(* IEC 61131-3 sources: IEC61131-3-CDSV3/Math Expressions Evaluator/src/20 Program Organization Units/_Internal, 7 files *)

(* ---- FuEvaluateFunctionCall.pou ---- *)
(*#-#-#-#-#-#-#-#-#-#---Declaration---#-#-#-#-#-#-#-#-#-#-#-#-#*)

// Evaluates a function call.
// First all necessary arguments are resolved to LREAL and then the function gets executed.
// The return value will indicate a successful evaluation.
{attribute 'qualified_only'}
FUNCTION INTERNAL FuEvaluateFunctionCall : BOOL
VAR_INPUT
    typFunctionToken: typExpressionToken;
    uiMaxCursor: UINT;
END_VAR
VAR_IN_OUT
    atTokens: ARRAY [*] OF typExpressionToken;
    uiCursor: UINT;

    alrVariables: ARRAY [*] OF LREAL;
    alrInternalVariables: ARRAY [*] OF LREAL;
END_VAR
VAR_OUTPUT
    lrResult: LREAL;
    sError: STRING;
END_VAR
{library PRIVATE}
VAR
    i: UINT;
    j: UINT;

    tempArgs: ARRAY [0..8] OF LREAL;
    tempHelperValue: LREAL;
END_VAR
VAR CONSTANT
    CONST_PI: LREAL := 3.14159265359;
END_VAR
(*#-#-#-#-#-#-#-#-#-#---Implementation---#-#-#-#-#-#-#-#-#-#-#-#-#*)

IF typFunctionToken.eType <> eTokenType.FUNCTION_CALL THEN
    sError := Standard.CONCAT('Invalid function call token at ', TO_STRING(uiCursor));
    RETURN;
END_IF

IF uiCursor + typFunctionToken.uiArgsCount > uiMaxCursor THEN
    sError := Standard.CONCAT('Not enough arguments for function call at ', TO_STRING(uiCursor));
    RETURN;
END_IF

FOR i := 0 TO (typFunctionToken.uiArgsCount - 1) BY 1 DO
    j := uiCursor + i + 1;

    IF NOT FuEvaluateTokenSingle(atTokens[j], j, alrVariables, alrInternalVariables, lrResult => tempArgs[i], sError => sError) THEN
        RETURN;
    END_IF
END_FOR

uiCursor := uiCursor + typFunctionToken.uiArgsCount;

IF typFunctionToken.sIdentifier = Constants.FUN_ABS THEN
    FuEvaluateFunctionCall := TRUE;
    lrResult := ABS(tempArgs[0]);
ELSIF typFunctionToken.sIdentifier = Constants.FUN_ACOS THEN
    FuEvaluateFunctionCall := TRUE;
    lrResult := ACOS(tempArgs[0]);
ELSIF typFunctionToken.sIdentifier = Constants.FUN_ASIN THEN
    FuEvaluateFunctionCall := TRUE;
    lrResult := ASIN(tempArgs[0]);
ELSIF typFunctionToken.sIdentifier = Constants.FUN_ATAN THEN
    FuEvaluateFunctionCall := TRUE;
    lrResult := ATAN(tempArgs[0]);
ELSIF typFunctionToken.sIdentifier = Constants.FUN_CEIL THEN
    FuEvaluateFunctionCall := TRUE;
    lrResult := FPU.Ceil(tempArgs[0]);
ELSIF typFunctionToken.sIdentifier = Constants.FUN_COS THEN
    FuEvaluateFunctionCall := TRUE;
    lrResult := COS(tempArgs[0]);
ELSIF typFunctionToken.sIdentifier = Constants.FUN_DEG THEN
    FuEvaluateFunctionCall := TRUE;
    lrResult := tempArgs[0] * 180 / CONST_PI;
ELSIF typFunctionToken.sIdentifier = Constants.FUN_FLOOR THEN
    FuEvaluateFunctionCall := TRUE;
    lrResult := FPU.Floor(tempArgs[0]);
ELSIF typFunctionToken.sIdentifier = Constants.FUN_LOG THEN
    FuEvaluateFunctionCall := TRUE;
    lrResult := LOG(tempArgs[0]);
ELSIF typFunctionToken.sIdentifier = Constants.FUN_LN THEN
    FuEvaluateFunctionCall := TRUE;
    lrResult := LN(tempArgs[0]);
ELSIF typFunctionToken.sIdentifier = Constants.FUN_RAD THEN
    FuEvaluateFunctionCall := TRUE;
    lrResult := tempArgs[0] * CONST_PI / 180;
ELSIF typFunctionToken.sIdentifier = Constants.FUN_ROUND THEN
    FuEvaluateFunctionCall := TRUE;

    IF (tempArgs[0] - FPU.Truncate(tempArgs[0])) >= 0.5 THEN
        lrResult := FPU.Ceil(tempArgs[0]);
    ELSE
        lrResult := FPU.Floor(tempArgs[0]);
    END_IF
ELSIF typFunctionToken.sIdentifier = Constants.FUN_SIN THEN
    FuEvaluateFunctionCall := TRUE;
    lrResult := SIN(tempArgs[0]);
ELSIF typFunctionToken.sIdentifier = Constants.FUN_SQRT THEN
    FuEvaluateFunctionCall := TRUE;
    lrResult := SQRT(tempArgs[0]);
ELSIF typFunctionToken.sIdentifier = Constants.FUN_TAN THEN
    FuEvaluateFunctionCall := TRUE;
    lrResult := TAN(tempArgs[0]);
ELSIF typFunctionToken.sIdentifier = Constants.FUN_TRUNC THEN
    FuEvaluateFunctionCall := TRUE;

    tempHelperValue := EXPT(10, tempArgs[1]);
    lrResult := FPU.Truncate((tempArgs[0] * tempHelperValue)) / tempHelperValue;
ELSIF typFunctionToken.sIdentifier = Constants.FUN_LIMIT THEN
    FuEvaluateFunctionCall := TRUE;
    lrResult := LIMIT(tempArgs[0], tempArgs[1], tempArgs[2]);
ELSIF typFunctionToken.sIdentifier = Constants.FUN_AVGA THEN
    FuEvaluateFunctionCall := TRUE;

    tempHelperValue := 0.0;
    FOR i := 0 TO (typFunctionToken.uiArgsCount - 1) BY 1 DO
        tempHelperValue := tempHelperValue + tempArgs[i];
    END_FOR

    lrResult := tempHelperValue / typFunctionToken.uiArgsCount;
ELSIF typFunctionToken.sIdentifier = Constants.FUN_MAX THEN
    FuEvaluateFunctionCall := TRUE;

    lrResult := -1.7976931348623157E+308;
    FOR i := 0 TO (typFunctionToken.uiArgsCount - 1) BY 1 DO
        IF tempArgs[i] > lrResult THEN
            lrResult := tempArgs[i];
        END_IF
    END_FOR
ELSIF typFunctionToken.sIdentifier = Constants.FUN_MIN THEN
    FuEvaluateFunctionCall := TRUE;

    lrResult := 1.7976931348623157E+308;
    FOR i := 0 TO (typFunctionToken.uiArgsCount - 1) BY 1 DO
        IF tempArgs[i] < lrResult THEN
            lrResult := tempArgs[i];
        END_IF
    END_FOR
ELSE
    sError := Standard.CONCAT('Function not implemented: ', typFunctionToken.sIdentifier);
END_IF

(* ---- FuEvaluateMathOp.pou ---- *)
(*#-#-#-#-#-#-#-#-#-#---Declaration---#-#-#-#-#-#-#-#-#-#-#-#-#*)

// Evaluates a math operation.
// First both tokens are resolved to LREAL values and then the selected operation takes place.
// In general, if any of the operands is a special LREAL value, then an error is returned.
// For Division (/), division by zero yields into an error (depends on ParameterList setting).
// For MODULO (%), both tokens are converted to LINT and the result is converted back to LREAL.
// The return value will indicate a successful evaluation.
{attribute 'qualified_only'}
FUNCTION INTERNAL FuEvaluateMathOp : BOOL
VAR_INPUT
    typOp: typExpressionToken;
    typToken1: typExpressionToken;
    typToken2: typExpressionToken;
    uiCursor: UINT;                  // Only for error message
END_VAR
VAR_IN_OUT
    alrVariables: ARRAY [*] OF LREAL;
    alrInternalVariables: ARRAY [*] OF LREAL;
END_VAR
VAR_OUTPUT
    lrResult: LREAL;
    sError: STRING;
END_VAR
{library PRIVATE}
VAR
    tempOperatorByte: BYTE;
    tempNumber1: LREAL;
    tempNumber2: LREAL;
END_VAR
(*#-#-#-#-#-#-#-#-#-#---Implementation---#-#-#-#-#-#-#-#-#-#-#-#-#*)

IF typOp.eType <> eTokenType.MATH_OP THEN
    sError := Standard.CONCAT('Invalid math operation token at ', TO_STRING(uiCursor));
    RETURN;
END_IF

// Change STRING identifier to BYTE (to match on FuTokenizeExpression strings)
tempOperatorByte := typOp.sIdentifier[0];

// Resolve first token to LREAL
IF NOT FuEvaluateTokenSingle(typToken1, uiCursor, alrVariables, alrInternalVariables, lrResult => tempNumber1, sError => sError) THEN
    FuEvaluateMathOp := FALSE;
    RETURN;
END_IF

// Resolve second token to LREAL
IF NOT FuEvaluateTokenSingle(typToken2, uiCursor, alrVariables, alrInternalVariables, lrResult => tempNumber2, sError => sError) THEN
    FuEvaluateMathOp := FALSE;
    RETURN;
END_IF

IF NOT FPU.IsLRealNumber(tempNumber1) THEN
    FuEvaluateMathOp := FALSE;
    sError := Standard.CONCAT('Special LREAL value is not valid: ', TO_STRING(tempNumber1));
    RETURN;
ELSIF NOT FPU.IsLRealNumber(tempNumber2) THEN
    FuEvaluateMathOp := FALSE;
    sError := Standard.CONCAT('Special LREAL value is not valid: ', TO_STRING(tempNumber2));
    RETURN;
END_IF

IF tempOperatorByte = Constants.CHAR_ADD THEN
    lrResult := tempNumber1 + tempNumber2;
ELSIF tempOperatorByte = Constants.CHAR_SUB THEN
    lrResult := tempNumber1 - tempNumber2;
ELSIF tempOperatorByte = Constants.CHAR_MUL THEN
    lrResult := tempNumber1 * tempNumber2;
ELSIF tempOperatorByte = Constants.CHAR_DIV THEN
    IF tempNumber2 = 0.0 THEN
        CASE ParameterList.eDivisionByZero OF
            eDivisionByZeroHandling.RESULT_IS_ZERO:
                FuEvaluateMathOp := TRUE;
                lrResult := 0.0;
                RETURN;

            eDivisionByZeroHandling.DIVISOR_IS_ONE:
                tempNumber2 := 1.0;
        ELSE
            sError := 'Division by zero is not allowed';
            RETURN;
        END_CASE
    END_IF

    lrResult := tempNumber1 / tempNumber2;
ELSIF tempOperatorByte = Constants.CHAR_MUL THEN
    lrResult := EXPT(tempNumber1, tempNumber2);
ELSIF tempOperatorByte = Constants.CHAR_MOD THEN
    lrResult := LINT_TO_LREAL((LREAL_TO_LINT(tempNumber1) MOD LREAL_TO_LINT(tempNumber2)));
ELSE
    sError := Standard.CONCAT('Not a variable token at position ', TO_STRING(uiCursor));
    RETURN;
END_IF

FuEvaluateMathOp := TRUE;

(* ---- FuEvaluateOperation.pou ---- *)
(*#-#-#-#-#-#-#-#-#-#---Declaration---#-#-#-#-#-#-#-#-#-#-#-#-#*)

// Evaluates an operation expression.
// For example "5 + 2", but not "5 + 2 + 1".
// The return value will indicate a successful evaluation.
{attribute 'qualified_only'}
FUNCTION FuEvaluateOperation : BOOL
VAR_INPUT
    uiMaxCursor: UINT;
END_VAR
VAR_IN_OUT
    atTokens: ARRAY [*] OF typExpressionToken;
    uiCursor: UINT;

    alrVariables: ARRAY [*] OF LREAL;
    alrInternalVariables: ARRAY [*] OF LREAL;
END_VAR
VAR_OUTPUT
    lrResult: LREAL;
    sError: STRING;
END_VAR
{library PRIVATE}
VAR
    tempLowerBound: UINT;
    tempUpperBound: UINT;

    tempToken1: typExpressionToken;
    tempToken2: typExpressionToken;
    tempToken3: typExpressionToken;

    tempVariableNr: UINT;
END_VAR
(*#-#-#-#-#-#-#-#-#-#---Implementation---#-#-#-#-#-#-#-#-#-#-#-#-#*)

tempLowerBound := TO_UINT(LOWER_BOUND(atTokens, 1));
tempUpperBound := MIN(uiMaxCursor, TO_UINT(UPPER_BOUND(atTokens, 1)));

tempToken1 := atTokens[uiCursor];

CASE tempToken1.eType OF
    eTokenType.INVALID, eTokenType.MATH_OP, eTokenType.GROUP_START, eTokenType.GROUP_END, eTokenType.FUNCTION_CALL_END:
        sError := Standard.CONCAT('Invalid token at position ', TO_STRING(uiCursor));
        RETURN;

    eTokenType.FUNCTION_CALL:
        FuEvaluateOperation := FuEvaluateFunctionCall(
            tempToken1,
            tempUpperBound,
            atTokens,
            uiCursor,
            alrVariables,
            alrInternalVariables,
            lrResult => lrResult,
            sError => sError
        );
        RETURN;
END_CASE

// If we're past the maximum position/cursor, evaluate the token (it should be a variable or number)
IF uiCursor = uiMaxCursor AND_THEN FuEvaluateTokenSingle(tempToken1, uiCursor, alrVariables, alrInternalVariables, lrResult => lrResult, sError => sError) THEN
    RETURN;
END_IF

uiCursor := uiCursor + 1;

// The first token wasn't a variable or number and we're out of bounds, error out
IF uiCursor > tempUpperBound THEN
    sError := 'Array upper bounds violation (not enough tokens)';
    RETURN;
END_IF

tempToken2 := atTokens[uiCursor];

CASE tempToken2.eType OF
    eTokenType.MATH_OP:
        uiCursor := uiCursor + 1;
        IF uiCursor > tempUpperBound THEN
            sError := 'Array upper bounds violation (not enough tokens)';
            RETURN;
        END_IF

        FuEvaluateOperation := FuEvaluateMathOp(
            tempToken2,
            tempToken1,
            atTokens[uiCursor],
            uiCursor,
            alrVariables,
            alrInternalVariables,
            lrResult => lrResult,
            sError => sError
        );
        RETURN;
ELSE
    sError := Standard.CONCAT('Invalid token at position ', TO_STRING(uiCursor));
    RETURN;
END_CASE

(* ---- FuEvaluateStep.pou ---- *)
(*#-#-#-#-#-#-#-#-#-#---Declaration---#-#-#-#-#-#-#-#-#-#-#-#-#*)

// Evaluates a single step.
// For multiple token "expressions" (i.e. "5 + 2 + 1"),
// the term will be evaluated left to right (in token order).
// The return value will indicate a successful expression evaluation.
{attribute 'qualified_only'}
FUNCTION FuEvaluateStep : BOOL
VAR_INPUT
    typStep: typExpressionStep;
END_VAR
VAR_OUTPUT
    lrResult: LREAL;
    sError: STRING;
END_VAR
VAR_IN_OUT
    alrVariables: ARRAY [*] OF LREAL;
    alrInternalVariables: ARRAY [*] OF LREAL;
END_VAR
{library PRIVATE}
VAR
    i: UINT;
    tempMaxCursor: UINT;
END_VAR
(*#-#-#-#-#-#-#-#-#-#---Implementation---#-#-#-#-#-#-#-#-#-#-#-#-#*)

IF typStep.uiCountTokens = 0 THEN
    FuEvaluateStep := TRUE;
    RETURN;
END_IF

lrResult := 0.0;
sError := '';

tempMaxCursor := typStep.uiCountTokens - 1;
FOR i := 0 TO tempMaxCursor BY 1 DO
    // For operations like "5 + 3 + 1", we need for the second step "+ 1"
    // to insert the previous result of "5 + 3", so we rewind one and overwrite it
    IF i > 0 AND_THEN typStep.atTokens[i].eType = eTokenType.MATH_OP THEN
        i := i - 1;
        typStep.atTokens[i].eType := eTokenType.NUMBER;
        typStep.atTokens[i].lrValue := lrResult;
    END_IF

    IF NOT FuEvaluateOperation(tempMaxCursor, typStep.atTokens, i, alrVariables, alrInternalVariables, lrResult => lrResult, sError => sError) THEN
        RETURN;
    END_IF
END_FOR

FuEvaluateStep := TRUE;

(* ---- FuEvaluateTokenSingle.pou ---- *)
(*#-#-#-#-#-#-#-#-#-#---Declaration---#-#-#-#-#-#-#-#-#-#-#-#-#*)

// Evaluates token types that are considered "single".
// This includes: numbers, variables, internal variables.
// The return value will indicate a successful evaluation.
{attribute 'qualified_only'}
FUNCTION INTERNAL FuEvaluateTokenSingle : BOOL
VAR_INPUT
    typToken: typExpressionToken;
    uiCursor: UINT;                  // Only for error message
END_VAR
VAR_IN_OUT
    alrVariables: ARRAY [*] OF LREAL;
    alrInternalVariables: ARRAY [*] OF LREAL;
END_VAR
VAR_OUTPUT
    lrResult: LREAL;
    sError: STRING;
END_VAR
{library PRIVATE}
VAR
    tempVariableNr: UINT;
END_VAR
(*#-#-#-#-#-#-#-#-#-#---Implementation---#-#-#-#-#-#-#-#-#-#-#-#-#*)

CASE typToken.eType OF
    eTokenType.NUMBER:
        FuEvaluateTokenSingle := TRUE;
        lrResult := typToken.lrValue;

    eTokenType.VARIABLE, eTokenType.INTERNAL_VAR:
        FuEvaluateTokenSingle := FuEvaluateVariable(typToken, uiCursor, alrVariables, alrInternalVariables, lrResult => lrResult, sError => sError);
ELSE
    sError := Standard.CONCAT('Invalid single token at position ', TO_STRING(uiCursor));
END_CASE

(* ---- FuEvaluateVariable.pou ---- *)
(*#-#-#-#-#-#-#-#-#-#---Declaration---#-#-#-#-#-#-#-#-#-#-#-#-#*)

// Evaluates variables and internal variables to their LREAL value.
// The return value will indicate a successful evaluation.
{attribute 'qualified_only'}
FUNCTION INTERNAL FuEvaluateVariable : BOOL
VAR_INPUT
    typToken: typExpressionToken;
    uiCursor: UINT;                  // Only for error message
END_VAR
VAR_IN_OUT
    alrVariables: ARRAY [*] OF LREAL;
    alrInternalVariables: ARRAY [*] OF LREAL;
END_VAR
VAR_OUTPUT
    lrResult: LREAL;
    sError: STRING;
END_VAR
{library PRIVATE}
VAR
    tempVariableNr: UINT;
END_VAR
(*#-#-#-#-#-#-#-#-#-#---Implementation---#-#-#-#-#-#-#-#-#-#-#-#-#*)

CASE typToken.eType OF
    eTokenType.VARIABLE:
        tempVariableNr := TO_UINT(typToken.lrValue);

        IF LOWER_BOUND(alrVariables, 1) <= tempVariableNr AND_THEN tempVariableNr <= UPPER_BOUND(alrVariables, 1) THEN
            FuEvaluateVariable := TRUE;
            lrResult := alrVariables[tempVariableNr];
        ELSE
            sError := Standard.CONCAT('Unknown variable ', TO_STRING(tempVariableNr));
        END_IF

    eTokenType.INTERNAL_VAR:
        tempVariableNr := TO_UINT(typToken.lrValue);

        IF LOWER_BOUND(alrInternalVariables, 1) <= tempVariableNr AND_THEN tempVariableNr <= UPPER_BOUND(alrInternalVariables, 1) THEN
            FuEvaluateVariable := TRUE;
            lrResult := alrInternalVariables[tempVariableNr];
        ELSE
            sError := Standard.CONCAT('Unknown internal variable ', TO_STRING(tempVariableNr));
        END_IF
ELSE
    sError := Standard.CONCAT('Not a variable token at position ', TO_STRING(uiCursor));
END_CASE

(* ---- FuInsertSortStepizeGroupFound.pou ---- *)
(*#-#-#-#-#-#-#-#-#-#---Declaration---#-#-#-#-#-#-#-#-#-#-#-#-#*)

// Slightly modified version of:
// https://forge.codesys.com/forge/talk/Runtime/thread/6ae1b1ff98/#31a5/f035/66da/5ba5/1553/b75d/ce46
//
// This version uses instead of basic datatypes a struct and sorts it by {group number} and then {token index}
{attribute 'qualified_only'}
FUNCTION INTERNAL FuInsertSortStepizeGroupFound : BOOL
VAR_INPUT
    pbBuffer: POINTER TO BYTE;                           // Pointer to buffer (array)
    diElements: DINT;                                    // Array length
END_VAR
{library PRIVATE}
VAR
    tempDataSize: UINT;                                  // Element size
    tempIndex: DINT;                                     // Loop index
    tempMinIndex: DINT;                                  // Loop lowest index tested
    tempMaxIndex: DINT;                                  // Loop highest index tested
    tempCurrentIndex: DINT;                              // Loop current tested element index
    tempTemp: ARRAY [1..8] OF BYTE;                      // Store temp value
    tempPtrElement1: POINTER TO typStepizeGroupFound;    // Pointer operator, current element
    tempPtrElement2: POINTER TO typStepizeGroupFound;    // Pointer operator, insert element
    tempElement1: typStepizeGroupFound;
    tempElement2: typStepizeGroupFound;
END_VAR
(*#-#-#-#-#-#-#-#-#-#---Implementation---#-#-#-#-#-#-#-#-#-#-#-#-#*)

tempDataSize := SIZEOF(typStepizeGroupFound);

FOR tempIndex := 1 TO diElements - 1 DO
    // Highest index tested
    tempMaxIndex := tempIndex;

    // Lowest index tested
    tempMinIndex := -1;

    // Element we need to insert
    tempPtrElement2 := pbBuffer + TO_UDINT(tempDataSize*tempIndex);

    REPEAT
        // Current test index
        tempCurrentIndex := tempMinIndex + (tempMaxIndex - tempMinIndex) / 2;

        // Get element at current test index
        tempPtrElement1 := pbBuffer + TO_UDINT(tempDataSize*tempCurrentIndex);

        // Test for ordering
        SysMem.SysMemCpy(pDest := ADR(tempElement1), pSrc := tempPtrElement1, udiCount := tempDataSize);
        SysMem.SysMemCpy(pDest := ADR(tempElement2), pSrc := tempPtrElement2, udiCount := tempDataSize);

        IF tempElement1.uiGroupNumber = tempElement2.uiGroupNumber THEN
            IF tempElement1.uiTokenIndex > tempElement2.uiTokenIndex THEN
                tempMaxIndex := tempCurrentIndex;
            ELSE
                tempMinIndex := tempCurrentIndex;
            END_IF
        ELSIF tempElement1.uiGroupNumber > tempElement2.uiGroupNumber THEN
            tempMaxIndex := tempCurrentIndex;
        ELSE
            tempMinIndex := tempCurrentIndex;
        END_IF
    UNTIL
        (tempMaxIndex - tempMinIndex) < 2
    END_REPEAT

    // Save value to insert
    SysMem.SysMemCpy(pDest := ADR(tempTemp), pSrc := tempPtrElement2, udiCount := tempDataSize);

    // Move block
    SysMem.SysMemMove(
        pDest := (pbBuffer + tempDataSize * (TO_UDINT(tempMaxIndex) + 1)),
        pSrc := (pbBuffer + TO_UDINT((tempDataSize * tempMaxIndex))),
        udiCount := (tempDataSize * TO_UDINT(tempIndex - tempMaxIndex))
    );

    // set key
    SysMem.SysMemCpy(pDest := (pbBuffer + tempDataSize * TO_UDINT(tempMaxIndex)), pSrc := ADR(tempTemp), udiCount := tempDataSize);
END_FOR

FuInsertSortStepizeGroupFound := TRUE;
